// TIA Portal V21 export
VAR_GLOBAL   // PLC tag table "ALARM BIT"
   "DOOR1 CLOSE PB BIT" AT %M145.0 : Bool;
   "PV BOILER TEMP" AT %MD146 : Real;
   "SET BOILER BIT" AT %M145.1 : Bool;
   "PLANT STEAM LOW BIT" AT %M145.2 : Bool;
   "PURE STEAM LOW BIT" AT %M145.3 : Bool;
   "COOLING WATER LOW BIT" AT %M145.4 : Bool;
   "DOOR1 SAFETY SENSOR BIT" AT %M145.5 : Bool;
   "DOOR2 SAFETY SENSOR BIT" AT %M145.6 : Bool;
   "BOILER WATER OK BIT" AT %M145.7 : Bool;
   "RESET C21" AT %M152.2 : Bool;
   "MAN BOILER INLET VAL" AT %M152.3 : Bool;
   RESET_c22 AT %M152.4 : Bool;
   PULSE63 AT %M152.5 : Bool;
   PULSE64 AT %M152.6 : Bool;
   "door2 allow" AT %M152.7 : Bool;
   Cham_exh_val_bit AT %M160.0 : Bool;
   pulse65 AT %M160.1 : Bool;
   "abort standard" AT %M160.2 : Bool;
   PULSE66 AT %M154.0 : Bool;
END_VAR
